(* Logix 5000 project; controller Transcat_L33ER vendor 1 type 14 code 107 rev 32.11; software revision 32.02; part 2 of 3 *)
(* tags used below, declared in another part *)
   AcsiiToReal1 : HexASCII_to_REAL;
   AllDevice1stScanDone : BOOL;   // When this bit is set - all devices have been scanned once and bits reset
   AllDeviceEnable : BOOL;   // A bit to enable or disable the running of all devices
   AllReset : BOOL;   // Bit to reset Auto/Man, AutoRun, RecipeRun, TimedRunEnable to 0 from PLC
   alwaysOFF : BOOL;
   AnyAutoRun : BOOL;   // Bit that in on if ANY device is placed into Auto run (to signal pre-start beed)
   AnyAutoRunFlag : BOOL;   // A flag that indicates if any device is in Auto Run (used with pre-start beep logic)
   AnyManRunFlag : BOOL;   // A flag that indicates if any device is in Manual Run (used with pre-start beep logic)
   AnyManualRun : BOOL;   // Bit that in on if ANY device is placed into manual run (to signal pre-start beed)
   Auto_Run_All_Interlock : BOOL;   // Bit to interlock all devices running in Auto
   Beep : BOOL;   // Bit to Activte Beacon Alarm
   ConversionError : BOOL;
   ConvertedFloat : REAL;
   CV_101_Output : ALIAS FOR TC_Remote_IO:5:O.1;   // CV_101 - 3 Way Valve - Recyle / Process
   Device : Device[20];
   DiscreteTemp : BOOL;   // A temporay boolean to hold positions during PLC transer
   dNum : INT;   // The index of the current device being processed
   DoseCounter : COUNTER;   // Counts the # of doses since last reset
   DoseCounterReset_HMI : BOOL;   // HMI bit to reset the dose counter
   DoseStart : BOOL;   // Bit to start dosing sequence
   DoseStartOneShot : BOOL;   // One shot to start dosing
   DoseStop : BOOL;   // Bit to stop dosing
   DoseStopOneShot : BOOL;   // one shot to stop dosing
   DoseTarget : REAL;   // Target dose amount
   FT103 : BronkhorstFlowMeter;
   FT104 : BronkhorstFlowMeter;
   FT105 : BronkhorstFlowMeter;
   GF201 : Thayer_WB_Feeder;   // Thayer 2 Tags
   GF201_Totalizer1 : ALIAS FOR Thayer2Data[9];   // Thayer 2 (GF201) Totalizer 1 in lbs
   GF201_Write_Total1Reset : ALIAS FOR Thayer2_BS:O.Data[2].1;   // Thayer 2 (GF1201) Totalizer 1 reset
   HMI_AllReset : BOOL;   // Bit to reset Auto/Man, AutoRun, RecipeRun, TimedRunEnable to 0 from HMI
   HMI_RecipeStart : BOOL;   // Bit to start and stop recipe from HMI
   InitCount : INT;   // Counter to cycle through each device on start-up and reset AutoMan, AutoRun, ManualRun bits
   NewDataToggle : BOOL;
   PT104_PV_RAW : ALIAS FOR TC_Remote_IO:1:I.Ch1Data;   // Raw (unscaled) pressure reading from PT104 - PSI * 100 (range 0 - 108 PSI)
   PT105_PV_RAW : ALIAS FOR TC_Remote_IO:1:I.Ch2Data;   // Raw (unscaled) pressure reading from PT105 - PSI * 100 (range 0 - 108 PSI)
   RecipeStart : BOOL;   // Bit to start and stop a recipe execution from PLC logic
   StartBeepTimer : TIMER;   // Timer to sound the beep alarm before starting a device
   TempHexIn : SINT[8];   // Place to copy 8 SINT for proessing by AOI
   TestBit1 : BOOL;   // Just a test bit - does not do anything
   Thayer2ResetTotal1_HMI : BOOL;   // Bit to reset Thayer2 - totalizer 1 from HMI
(* MainProgram, continued *)

ROUTINE _08_FT104_Water_Dosing   (* ladder *)
// FT104 Control Logic not associated with Device Iteration Logic
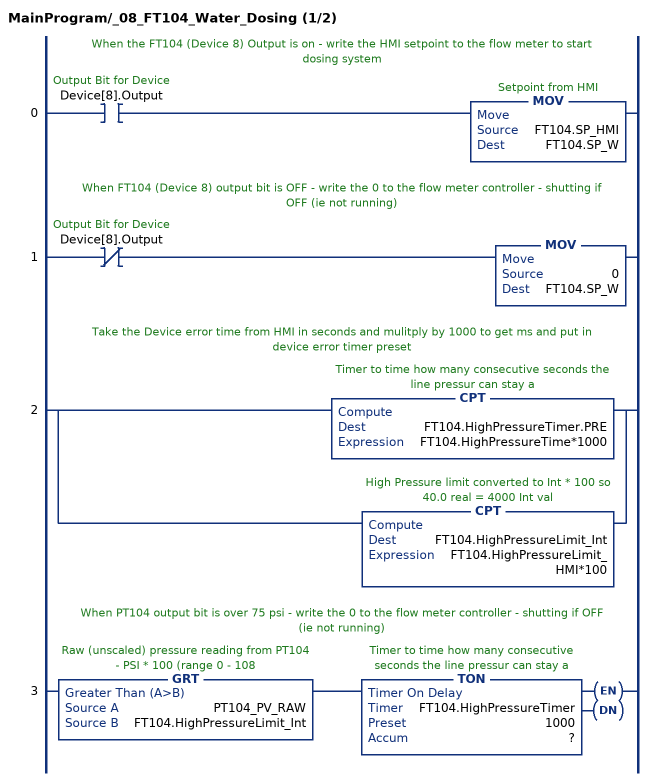
   // When the FT104 (Device 8) Output is on - write the HMI setpoint to the flow meter to start dosing system
   0: XIC(Device[8].Output)MOV(FT104.SP_HMI,FT104.SP_W);
   // When FT104 (Device 8) output bit is OFF - write the 0 to the flow meter controller - shutting if OFF (ie not running)
   1: XIO(Device[8].Output)MOV(0,FT104.SP_W);
   // Take the Device error time from HMI in seconds and mulitply by 1000 to get ms and put in  device error timer preset
   2: [CPT(FT104.HighPressureTimer.PRE,FT104.HighPressureTime*1000) ,CPT(FT104.HighPressureLimit_Int,FT104.HighPressureLimit_HMI*100) ];
   // When PT104 output bit is over 75 psi - write the 0 to the flow meter controller - shutting if OFF (ie not running)
   3: GRT(PT104_PV_RAW,FT104.HighPressureLimit_Int)TON(FT104.HighPressureTimer,?,?);
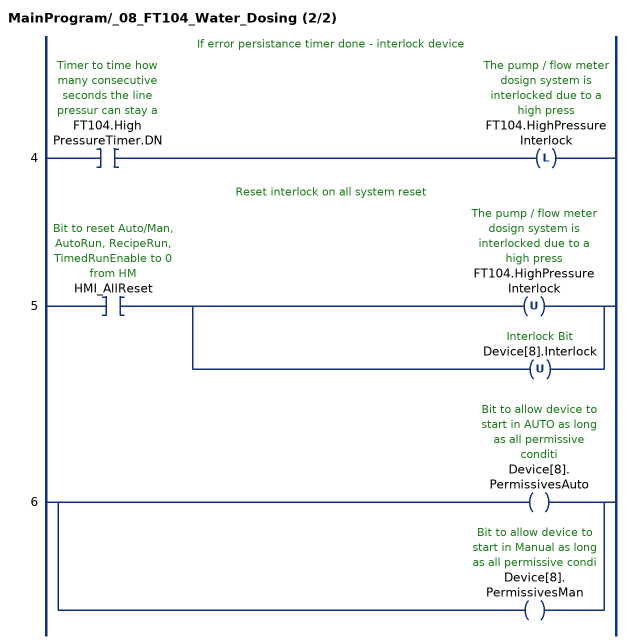
   // If error persistance timer done - interlock device
   4: XIC(FT104.HighPressureTimer.DN)OTL(FT104.HighPressureInterlock);
   // Reset interlock on all system reset
   5: XIC(HMI_AllReset)[OTU(FT104.HighPressureInterlock) ,OTU(Device[8].Interlock) ];
   6: [OTE(Device[8].PermissivesAuto) ,OTE(Device[8].PermissivesMan) ];
END_ROUTINE

ROUTINE _09_FT105_Fragrance_Dosing   (* ladder *)
// FT105 Control Logic not associated with Device Iteration Logic
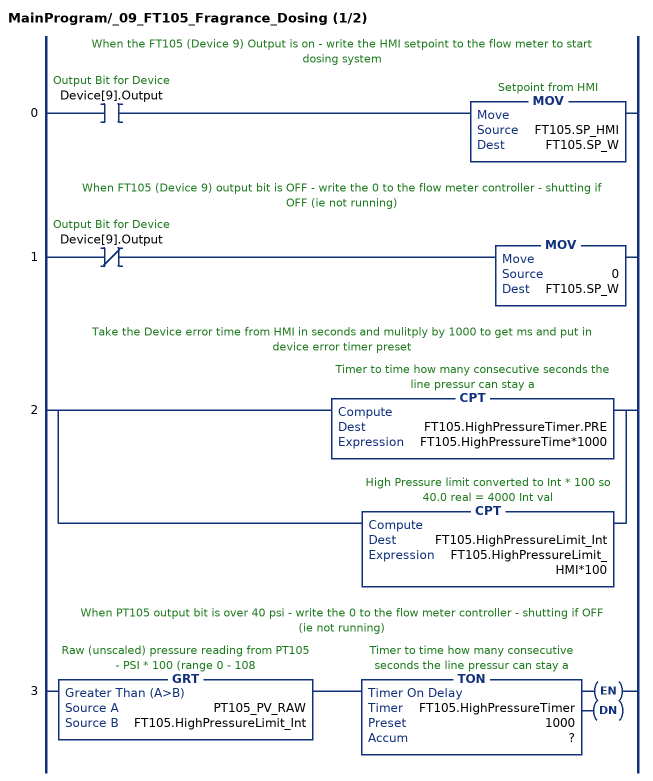
   // When the FT105 (Device 9) Output is on - write the HMI setpoint to the flow meter to start dosing system
   0: XIC(Device[9].Output)MOV(FT105.SP_HMI,FT105.SP_W);
   // When FT105 (Device 9) output bit is OFF - write the 0 to the flow meter controller - shutting if OFF (ie not running)
   1: XIO(Device[9].Output)MOV(0,FT105.SP_W);
   // Take the Device error time from HMI in seconds and mulitply by 1000 to get ms and put in  device error timer preset
   2: [CPT(FT105.HighPressureTimer.PRE,FT105.HighPressureTime*1000) ,CPT(FT105.HighPressureLimit_Int,FT105.HighPressureLimit_HMI*100) ];
   // When PT105 output bit is over 40 psi - write the 0 to the flow meter controller - shutting if OFF (ie not running)
   3: GRT(PT105_PV_RAW,FT105.HighPressureLimit_Int)TON(FT105.HighPressureTimer,?,?);
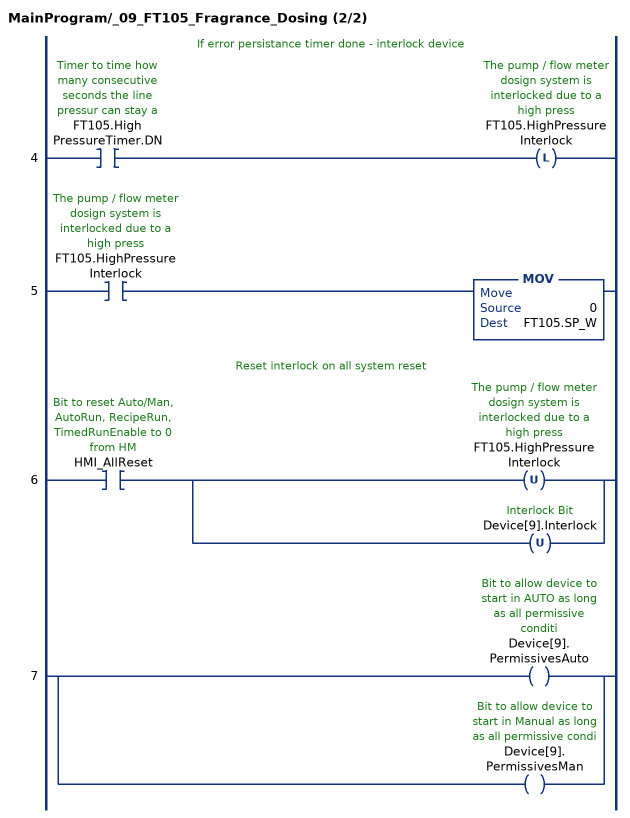
   // If error persistance timer done - interlock device
   4: XIC(FT105.HighPressureTimer.DN)OTL(FT105.HighPressureInterlock);
   5: XIC(FT105.HighPressureInterlock)MOV(0,FT105.SP_W);
   // Reset interlock on all system reset
   6: XIC(HMI_AllReset)[OTU(FT105.HighPressureInterlock) ,OTU(Device[9].Interlock) ];
   7: [OTE(Device[9].PermissivesAuto) ,OTE(Device[9].PermissivesMan) ];
END_ROUTINE

ROUTINE _11_Auxillary_Pump_AE   (* ladder *)
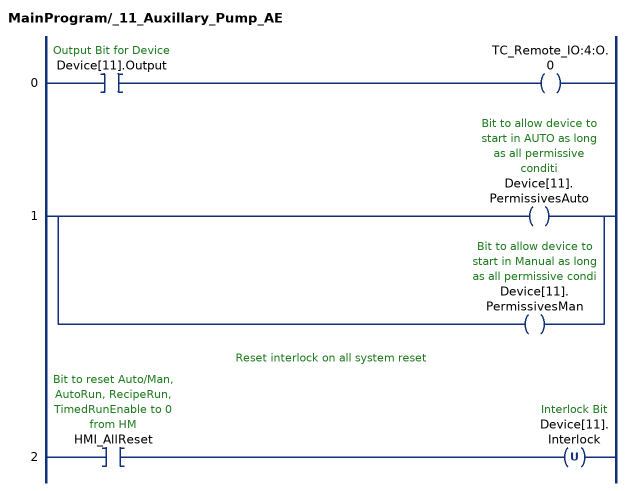
   0: XIC(Device[11].Output)OTE(TC_Remote_IO:4:O.0);
   1: [OTE(Device[11].PermissivesAuto) ,OTE(Device[11].PermissivesMan) ];
   // Reset interlock on all system reset
   2: XIC(HMI_AllReset)OTU(Device[11].Interlock);
END_ROUTINE

ROUTINE _12_SC_1_Screener   (* ladder *)
// Screener
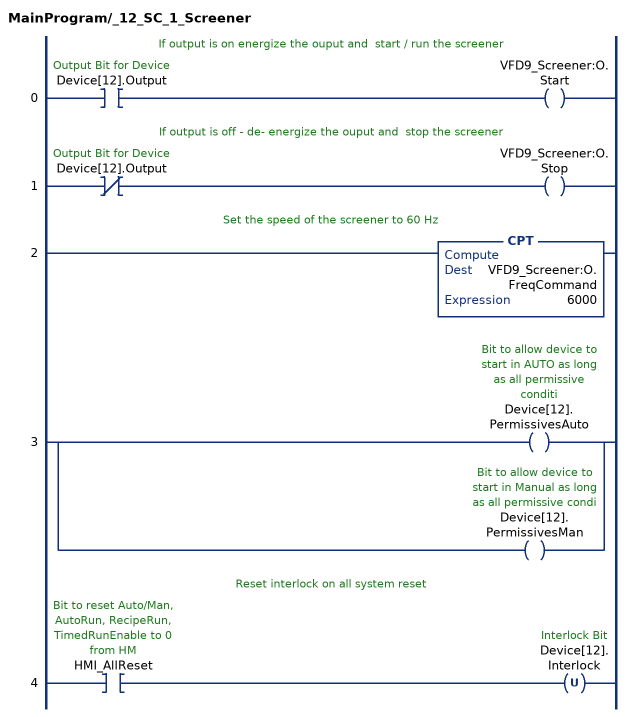
   // If output is on energize the ouput and  start / run the screener
   0: XIC(Device[12].Output)OTE(VFD9_Screener:O.Start);
   // If output is off - de- energize the ouput and  stop the screener
   1: XIO(Device[12].Output)OTE(VFD9_Screener:O.Stop);
   // Set the speed of the screener to 60 Hz
   2: CPT(VFD9_Screener:O.FreqCommand,6000);
   3: [OTE(Device[12].PermissivesAuto) ,OTE(Device[12].PermissivesMan) ];
   // Reset interlock on all system reset
   4: XIC(HMI_AllReset)OTU(Device[12].Interlock);
END_ROUTINE

ROUTINE _13_CV101_3_Way_Dosing_Value   (* ladder *)
// 3 way valve to switch between recyle and feed to process
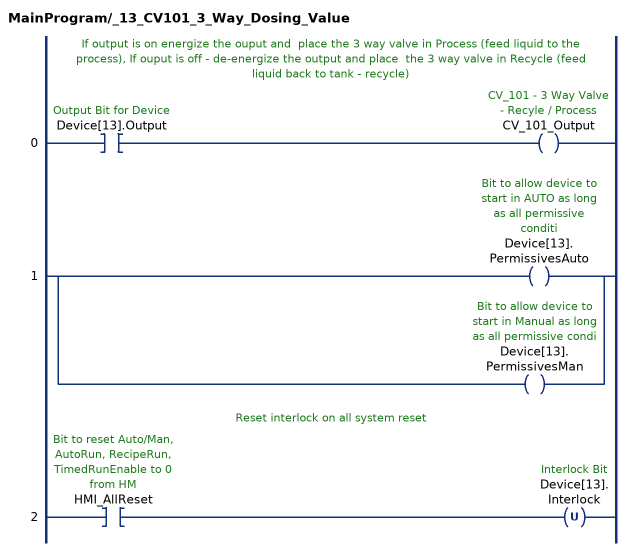
   // If output is on energize the ouput and  place the 3 way valve in Process (feed liquid to the process), If ouput is off - de-energize the output and place  the 3 way valve in Recycle (feed liquid back to tank - recycle)
   0: XIC(Device[13].Output)OTE(CV_101_Output);
   1: [OTE(Device[13].PermissivesAuto) ,OTE(Device[13].PermissivesMan) ];
   // Reset interlock on all system reset
   2: XIC(HMI_AllReset)OTU(Device[13].Interlock);
END_ROUTINE

ROUTINE Bronkhorst_Data   (* ladder *)
// read and write data to/from the EIP instance and convert to/from 8 byte to/from floating point
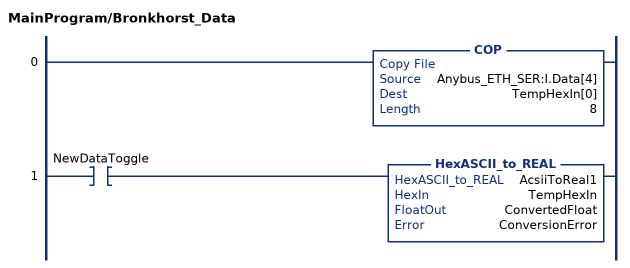
   0: COP(Anybus_ETH_SER:I.Data[4],TempHexIn[0],8);
   1: XIC(NewDataToggle)HexASCII_to_REAL(AcsiiToReal1,TempHexIn,ConvertedFloat,ConversionError);
END_ROUTINE

ROUTINE DeviceLogic   (* ladder *)
// Process the logic for each device with index and indirect addressing.
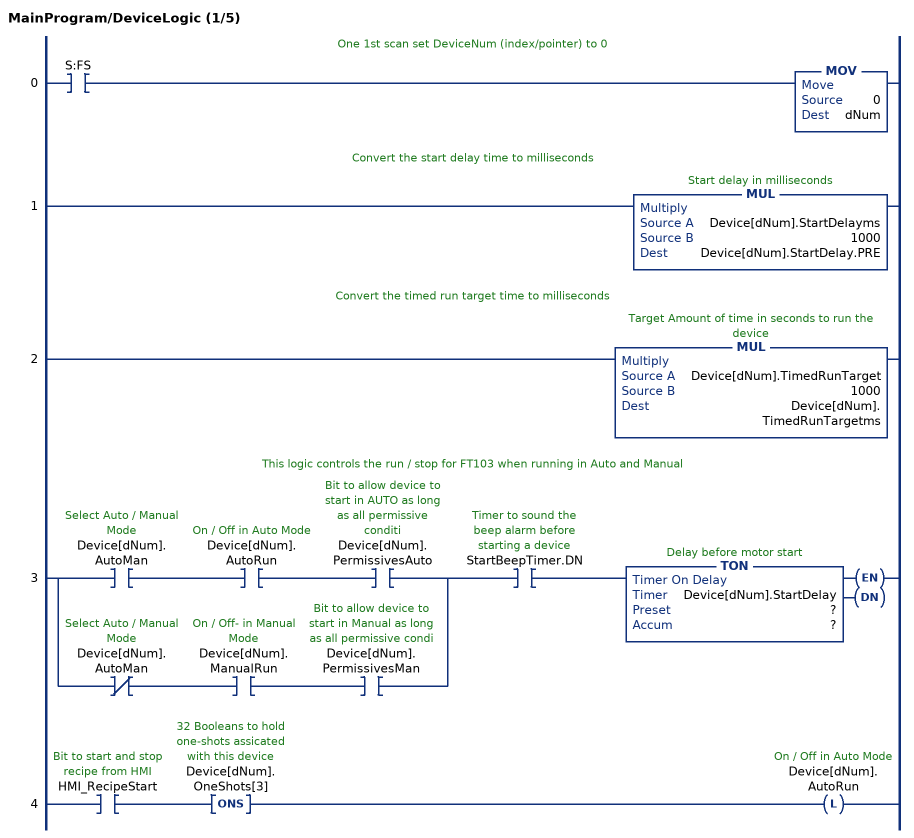
   // One 1st scan set DeviceNum (index/pointer) to 0
   0: XIC(S:FS)MOV(0,dNum);
   // Convert the start delay time to milliseconds
   1: MUL(Device[dNum].StartDelayms,1000,Device[dNum].StartDelay.PRE);
   // Convert the timed run target time to milliseconds
   2: MUL(Device[dNum].TimedRunTarget,1000,Device[dNum].TimedRunTargetms);
   // This logic controls the run / stop for FT103 when running in Auto and Manual
   3: [XIC(Device[dNum].AutoMan) XIC(Device[dNum].AutoRun) XIC(Device[dNum].PermissivesAuto) ,XIO(Device[dNum].AutoMan) XIC(Device[dNum].ManualRun) XIC(Device[dNum].PermissivesMan) ]XIC(StartBeepTimer.DN)TON(Device[dNum].StartDelay,?,?);
   4: XIC(HMI_RecipeStart)ONS(Device[dNum].OneShots[3])OTL(Device[dNum].AutoRun);
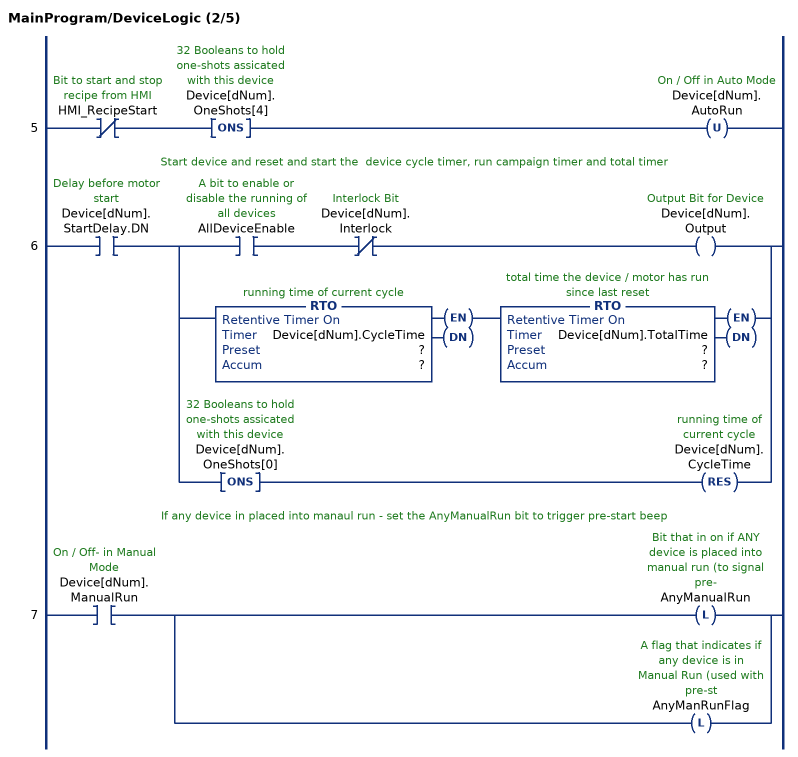
   5: XIO(HMI_RecipeStart)ONS(Device[dNum].OneShots[4])OTU(Device[dNum].AutoRun);
   // Start device and reset and start the  device cycle timer, run campaign timer and total timer
   6: XIC(Device[dNum].StartDelay.DN)[XIC(AllDeviceEnable) XIO(Device[dNum].Interlock) OTE(Device[dNum].Output) ,[RTO(Device[dNum].CycleTime,?,?) RTO(Device[dNum].TotalTime,?,?) ,ONS(Device[dNum].OneShots[0]) RES(Device[dNum].CycleTime) ] ];
   // If any device in placed into manaul run - set the AnyManualRun bit to trigger pre-start beep
   7: XIC(Device[dNum].ManualRun)[OTL(AnyManualRun) ,OTL(AnyManRunFlag) ];
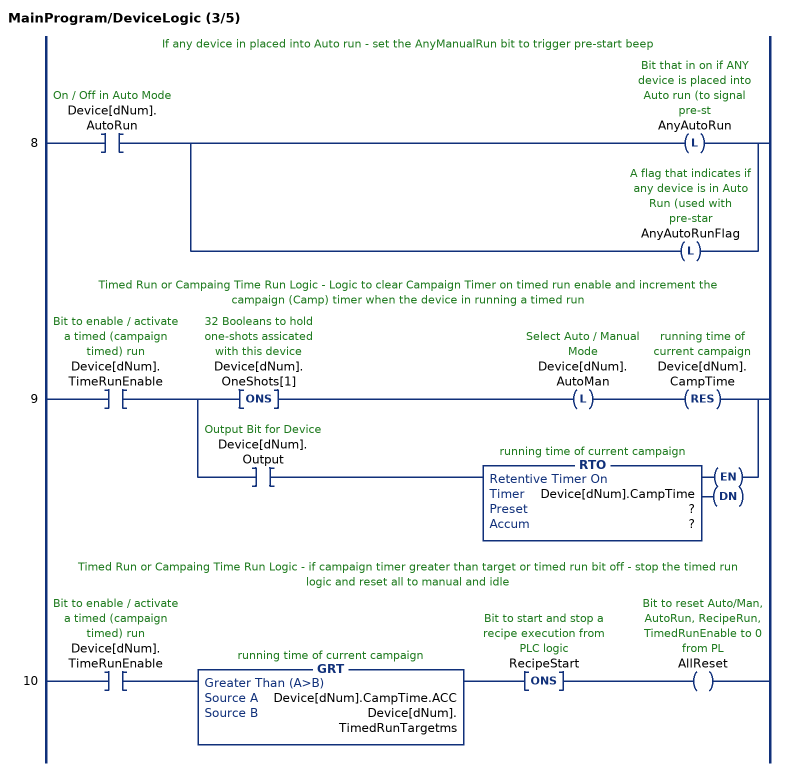
   // If any device in placed into Auto run - set the AnyManualRun bit to trigger pre-start beep
   8: XIC(Device[dNum].AutoRun)[OTL(AnyAutoRun) ,OTL(AnyAutoRunFlag) ];
   // Timed Run or Campaing Time Run Logic - Logic to clear Campaign Timer on timed run enable and increment the campaign (Camp) timer when the device in running a timed run
   9: XIC(Device[dNum].TimeRunEnable)[ONS(Device[dNum].OneShots[1]) OTL(Device[dNum].AutoMan) RES(Device[dNum].CampTime) ,XIC(Device[dNum].Output) RTO(Device[dNum].CampTime,?,?) ];
   // Timed Run or Campaing Time Run Logic - if campaign timer greater than target or timed run bit off - stop the timed run logic and reset all to manual and idle
   10: XIC(Device[dNum].TimeRunEnable)GRT(Device[dNum].CampTime.ACC,Device[dNum].TimedRunTargetms)ONS(RecipeStart)OTE(AllReset);
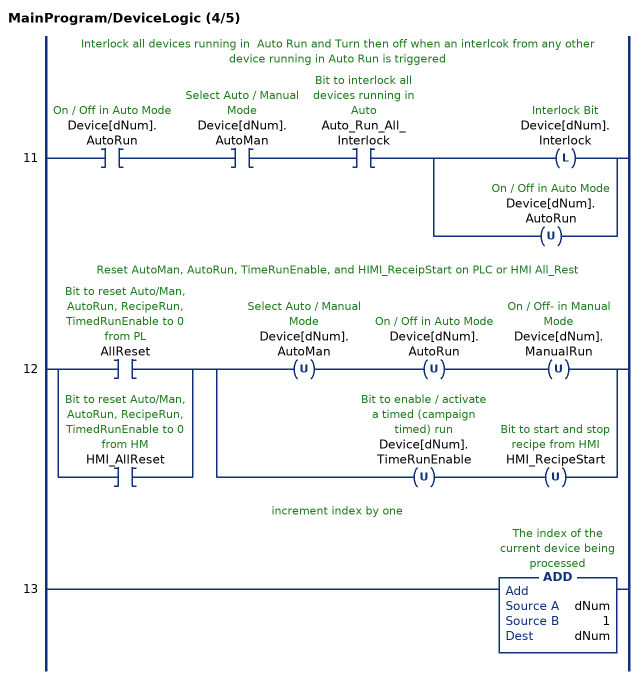
   // Interlock all devices running in  Auto Run and Turn then off when an interlcok from any other device running in Auto Run is triggered
   11: XIC(Device[dNum].AutoRun)XIC(Device[dNum].AutoMan)XIC(Auto_Run_All_Interlock)[OTL(Device[dNum].Interlock) ,OTU(Device[dNum].AutoRun) ];
   // Reset AutoMan, AutoRun, TimeRunEnable, and HIMI_ReceipStart on PLC or HMI All_Rest
   12: [XIC(AllReset) ,XIC(HMI_AllReset) ][OTU(Device[dNum].AutoMan) OTU(Device[dNum].AutoRun) OTU(Device[dNum].ManualRun) ,OTU(Device[dNum].TimeRunEnable) OTU(HMI_RecipeStart) ];
   // increment index by one
   13: ADD(dNum,1,dNum);
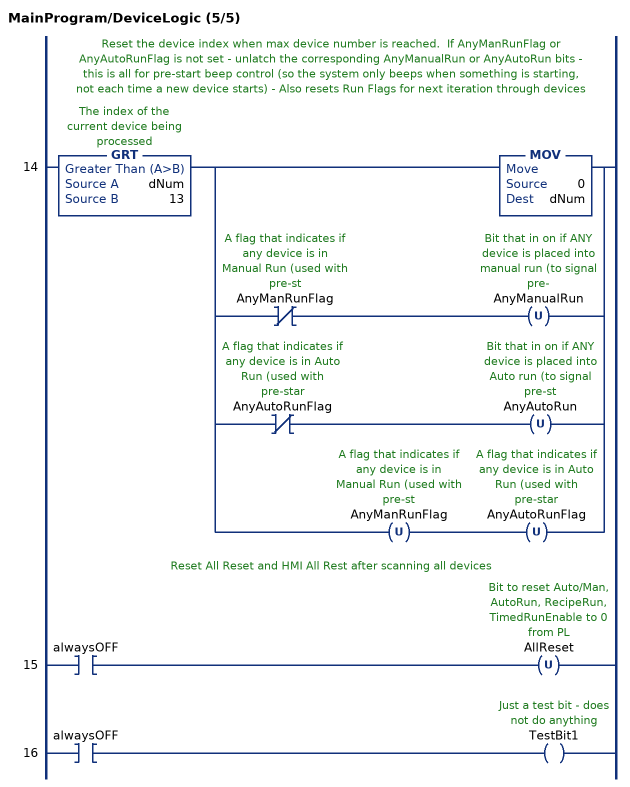
   // Reset the device index when max device number is reached.  If AnyManRunFlag or AnyAutoRunFlag is not set - unlatch the corresponding AnyManualRun or AnyAutoRun bits - this is all for pre-start beep control (so the system only beeps when something is starting, not each time a new device starts) - Also resets Run Flags for next iteration through devices
   14: GRT(dNum,13)[[MOV(0,dNum) ,[XIO(AnyManRunFlag) OTU(AnyManualRun) ,XIO(AnyAutoRunFlag) OTU(AnyAutoRun) ] ] ,OTU(AnyManRunFlag) OTU(AnyAutoRunFlag) ];
   // Reset All Reset and HMI All Rest after scanning all devices
   15: XIC(alwaysOFF)OTU(AllReset);
   16: XIC(alwaysOFF)OTE(TestBit1);
END_ROUTINE

ROUTINE GF201Dose   (* ladder *)
// Logic to Dose a specific amount from GF201 - Thayer 2
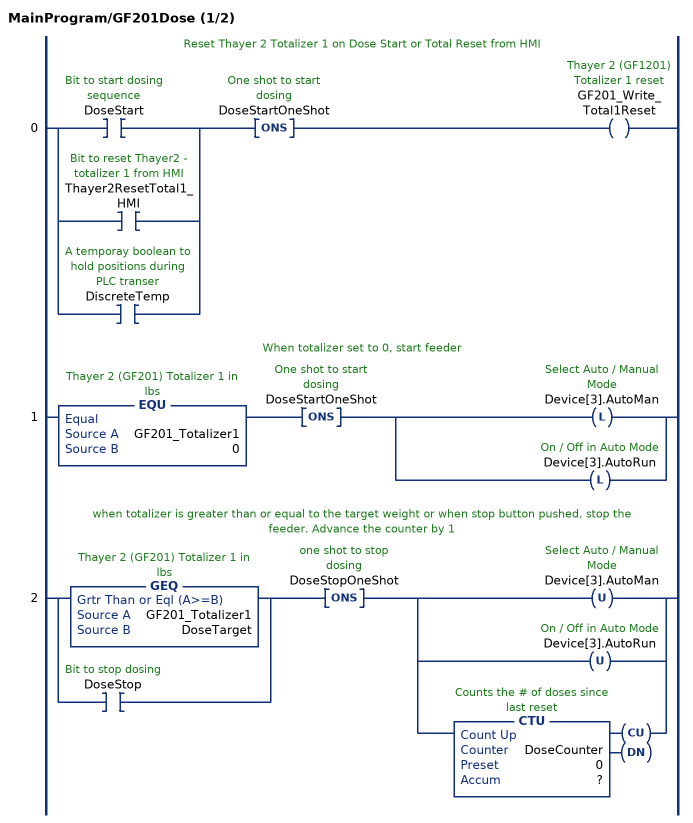
   // Reset Thayer 2 Totalizer 1 on Dose Start or Total Reset from HMI
   0: [XIC(DoseStart) ,[XIC(Thayer2ResetTotal1_HMI) ,XIC(DiscreteTemp) ] ]ONS(DoseStartOneShot)OTE(GF201_Write_Total1Reset);
   // When totalizer set to 0, start feeder
   1: EQU(GF201_Totalizer1,0)ONS(DoseStartOneShot)[OTL(Device[3].AutoMan) ,OTL(Device[3].AutoRun) ];
   // when totalizer is greater than or equal to the target weight or when stop button pushed, stop the feeder. Advance the counter by 1
   2: [GEQ(GF201_Totalizer1,DoseTarget) ,XIC(DoseStop) ]ONS(DoseStopOneShot)[OTU(Device[3].AutoMan) ,[OTU(Device[3].AutoRun) ,CTU(DoseCounter,?,?) ] ];
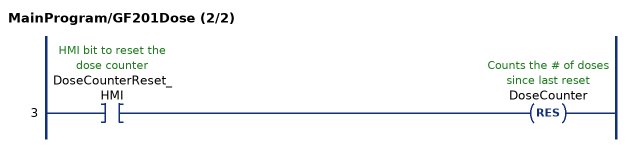
   3: XIC(DoseCounterReset_HMI)RES(DoseCounter);
END_ROUTINE

ROUTINE Initialize   (* ladder *)
// Reset controls and any other initialization required
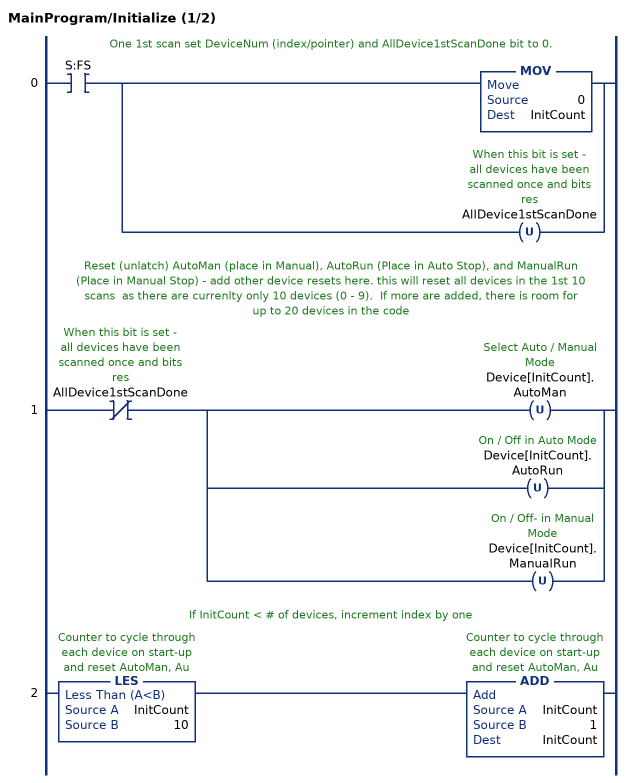
   // One 1st scan set DeviceNum (index/pointer) and AllDevice1stScanDone bit to 0.
   0: XIC(S:FS)[MOV(0,InitCount) ,OTU(AllDevice1stScanDone) ];
   // Reset (unlatch) AutoMan (place in Manual), AutoRun (Place in Auto Stop), and ManualRun (Place in Manual Stop) - add other device resets here. this will reset all devices in the 1st 10 scans  as there are currenlty only 10 devices (0 - 9).  If more are added, there is room for up to 20 devices in the code
   1: XIO(AllDevice1stScanDone)[OTU(Device[InitCount].AutoMan) ,[OTU(Device[InitCount].AutoRun) ,OTU(Device[InitCount].ManualRun) ] ];
   // If InitCount < # of devices, increment index by one
   2: LES(InitCount,10)ADD(InitCount,1,InitCount);
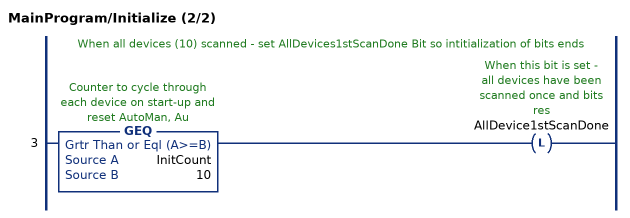
   // When all devices (10) scanned - set AllDevices1stScanDone Bit so intitialization of bits ends
   3: GEQ(InitCount,10)OTL(AllDevice1stScanDone);
END_ROUTINE

ROUTINE InterlockLogic   (* ladder *)
// All interlock logic is handled here
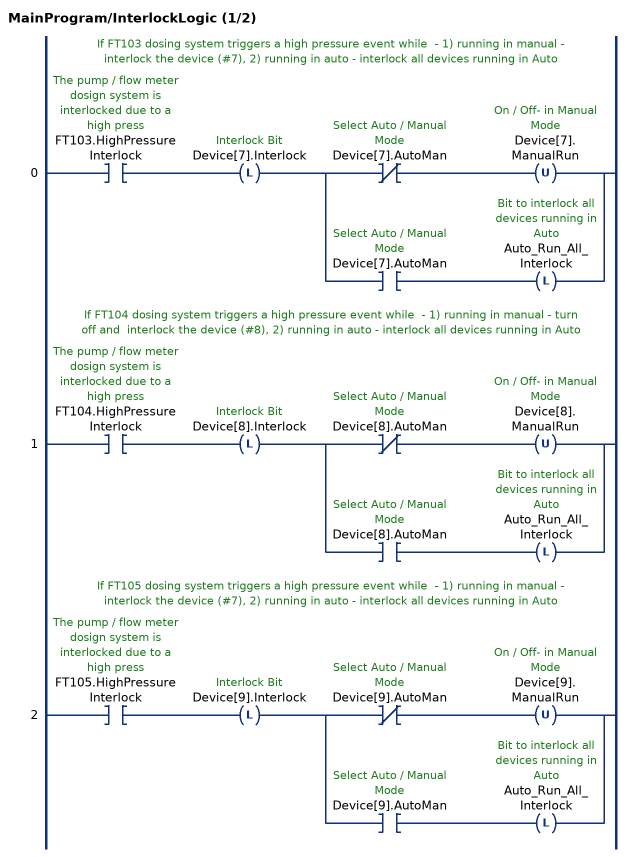
   // If FT103 dosing system triggers a high pressure event while  - 1) running in manual - interlock the device (#7), 2) running in auto - interlock all devices running in Auto
   0: XIC(FT103.HighPressureInterlock)OTL(Device[7].Interlock)[XIO(Device[7].AutoMan) OTU(Device[7].ManualRun) ,XIC(Device[7].AutoMan) OTL(Auto_Run_All_Interlock) ];
   // If FT104 dosing system triggers a high pressure event while  - 1) running in manual - turn off and  interlock the device (#8), 2) running in auto - interlock all devices running in Auto
   1: XIC(FT104.HighPressureInterlock)OTL(Device[8].Interlock)[XIO(Device[8].AutoMan) OTU(Device[8].ManualRun) ,XIC(Device[8].AutoMan) OTL(Auto_Run_All_Interlock) ];
   // If FT105 dosing system triggers a high pressure event while  - 1) running in manual - interlock the device (#7), 2) running in auto - interlock all devices running in Auto
   2: XIC(FT105.HighPressureInterlock)OTL(Device[9].Interlock)[XIO(Device[9].AutoMan) OTU(Device[9].ManualRun) ,XIC(Device[9].AutoMan) OTL(Auto_Run_All_Interlock) ];
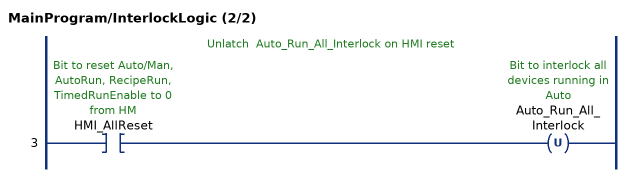
   // Unlatch  Auto_Run_All_Interlock on HMI reset
   3: XIC(HMI_AllReset)OTU(Auto_Run_All_Interlock);
END_ROUTINE
